// TIA Portal V21 export
DATA_BLOCK "Mm01Mixing"   // DB306
AUTHOR : PRECISE
FAMILY : PRECISE
// stored: AutoNumber false, InstanceOfName FB302, InstanceOfType FB
"FB302"
   // VAR_INPUT
   //    Enable : Bool;
   //    Disable : Bool;
   //    Fault : Bool;
   //    SecPulse : Bool;
   //    AlwaysTrue : Bool;
   //    StartConfirmationPopupSel : Bool;
   //    EndConfirmationPopupSel : Bool;
   //    MixingModeSel : Int;
   //    MixerTypeSel : Int := 4;
   //    MixingTimeBaseSel : Bool := 1;
   //    MixingTimeMin : Int;
   //    MixingTimeSec : Int;
   //    MixingSpeed : Real;
   // END_VAR
   // VAR_OUTPUT
   //    MixerCmd : Bool;
   //    WaterInletValve : Bool;
   //    StartConfirmationPopup : Bool;
   //    EndConfirmationPopup : Bool;
   //    ManualPopup : Bool;
   //    MixingTimeMinPV : DInt;
   //    MixingTimeSecPV : DInt;
   //    MixingSpeedPV : Real;
   //    PrintTrigger : Bool;
   //    PrintWord : Int;
   //    PrintStatus : String[50];
   // END_VAR
   // VAR_IN_OUT
   //    Start : Bool;
   //    Stop : Bool;
   //    Reset : Bool;
   //    StartConfirmationAck : Bool;
   //    EndConfirmationAck : Bool;
   //    ManualAck : Bool;
   //    Cp01Fsc : Bool;
   //    SpareBtn2 : Bool;
   //    Running : Bool;
   //    Selected : Bool;
   //    Paused : Bool;
   //    StartConfirmationPopupTemp : Bool;
   //    EndConfirmationPopupTemp : Bool;
   //    ManualPopupTemp : Bool;
   //    MixingStarted : Bool;
   //    MixingOver : Bool;
   // END_VAR
   // VAR
   //    PrintTriggerTemp : Bool;
   //    RE1 : Bool;
   //    RE2 : Bool;
   //    RE3 : Bool;
   //    RE4 : Bool;
   //    RE5 : Bool;
   //    RE6 : Bool;
   //    RE7 : Bool;
   //    MixingTimer : "FB101";
   //    PrintTriggerResetTimer { S7_SetPoint := 'True'} : TON_TIME;
   //    BtnResetTimer { S7_SetPoint := 'True'} : TON_TIME;
   // END_VAR
BEGIN
END_DATA_BLOCK
